SYSTEM Example System
  (* Version 1.0, 2007-08-28, Goran, Chalmers *)
  DEVICE Test Device : DeviceType_not_used
    RESOURCE TestResource : ResourceType_not_used
      FBS
        restart : E_RESTART;
        stop : E_STOP;
        split : E_SPLIT2;
        rend : E_REND;
        prod1 : Product;
        prod2 : Product;
        res1 : Resource;
        res2 : Resource;
        res3 : Resource;
        mux1take : Mux;
        mux1process : Mux;
        mux1release : Mux;
        mux2take : Mux;
        mux2process : Mux;
        mux2release : Mux;
        mux3take : Mux;
        mux3process : Mux;
        mux3release : Mux;
        datamux1 : DataMux;
        datamux2 : DataMux;
        datamux3 : DataMux;
        datademux1 : DataDemux;
        datademux2 : DataDemux;
        datademux3 : DataDemux;
        demux1taken : Demux;
        demux1processed : Demux;
        demux2taken : Demux;
        demux2processed : Demux;
        demux3taken : Demux;
        demux3processed : Demux;
      END_FBS
      EVENT_CONNECTIONS
        restart.COLD TO split.EI;
        split.EO1 TO prod1.make;
        split.EO2 TO prod2.make;
        prod1.takeR1 TO mux1take.EI1;
        prod1.processR1 TO mux1process.EI1;
        prod1.releaseR1 TO mux1release.EI1;
        prod2.takeR1 TO mux1take.EI2;
        prod2.processR1 TO mux1process.EI2;
        prod2.releaseR1 TO mux1release.EI2;
        mux1take.EO TO datamux1.EI1;
        mux1process.EO TO datamux1.EI2;
        mux1release.EO TO datamux1.EI3;
        datamux1.EO1 TO res1.take;
        datamux1.EO2 TO res1.process;
        datamux1.EO3 TO res1.release;
        res1.taken TO datademux1.EI1;
        res1.processed TO datademux1.EI2;
        datademux1.EO1 TO demux1taken.EI;
        datademux1.EO2 TO demux1processed.EI;
        demux1taken.EO1 TO prod1.gotR1;
        demux1taken.EO2 TO prod2.gotR1;
        demux1processed.EO1 TO prod1.processedR1;
        demux1processed.EO2 TO prod2.processedR1;
        prod1.takeR2 TO mux2take.EI1;
        prod1.processR2 TO mux2process.EI1;
        prod1.releaseR2 TO mux2release.EI1;
        prod2.takeR2 TO mux2take.EI2;
        prod2.processR2 TO mux2process.EI2;
        prod2.releaseR2 TO mux2release.EI2;
        mux2take.EO TO datamux2.EI1;
        mux2process.EO TO datamux2.EI2;
        mux2release.EO TO datamux2.EI3;
        datamux2.EO1 TO res2.take;
        datamux2.EO2 TO res2.process;
        datamux2.EO3 TO res2.release;
        res2.taken TO datademux2.EI1;
        res2.processed TO datademux2.EI2;
        datademux2.EO1 TO demux2taken.EI;
        datademux2.EO2 TO demux2processed.EI;
        demux2taken.EO1 TO prod1.gotR2;
        demux2taken.EO2 TO prod2.gotR2;
        demux2processed.EO1 TO prod1.processedR2;
        demux2processed.EO2 TO prod2.processedR2;
        prod1.takeR3 TO mux3take.EI1;
        prod1.processR3 TO mux3process.EI1;
        prod1.releaseR3 TO mux3release.EI1;
        prod2.takeR3 TO mux3take.EI2;
        prod2.processR3 TO mux3process.EI2;
        prod2.releaseR3 TO mux3release.EI2;
        mux3take.EO TO datamux3.EI1;
        mux3process.EO TO datamux3.EI2;
        mux3release.EO TO datamux3.EI3;
        datamux3.EO1 TO res3.take;
        datamux3.EO2 TO res3.process;
        datamux3.EO3 TO res3.release;
        res3.taken TO datademux3.EI1;
        res3.processed TO datademux3.EI2;
        datademux3.EO1 TO demux3taken.EI;
        datademux3.EO2 TO demux3processed.EI;
        demux3taken.EO1 TO prod1.gotR3;
        demux3taken.EO2 TO prod2.gotR3;
        demux3processed.EO1 TO prod1.processedR3;
        demux3processed.EO2 TO prod2.processedR3;
        prod1.done TO rend.EI1;
        prod2.done TO rend.EI2;
        rend.EO TO stop.STOP;
      END_CONNECTIONS
      DATA_CONNECTIONS
        1 TO prod1.product;
        2 TO prod2.product;
        1 TO res1.capacity;
        1 TO res2.capacity;
        1 TO res3.capacity;
        mux1take.DO TO datamux1.DI1;
        mux1process.DO TO datamux1.DI2;
        mux1release.DO TO datamux1.DI3;
        datamux1.DO TO res1.product;
        res1.forProduct TO datademux1.DI;
        datademux1.DO1 TO demux1taken.DI;
        datademux1.DO2 TO demux1processed.DI;
        mux2take.DO TO datamux2.DI1;
        mux2process.DO TO datamux2.DI2;
        mux2release.DO TO datamux2.DI3;
        datamux2.DO TO res2.product;
        res2.forProduct TO datademux2.DI;
        datademux2.DO1 TO demux2taken.DI;
        datademux2.DO2 TO demux2processed.DI;
        mux3take.DO TO datamux3.DI1;
        mux3process.DO TO datamux3.DI2;
        mux3release.DO TO datamux3.DI3;
        datamux3.DO TO res3.product;
        res3.forProduct TO datademux3.DI;
        datademux3.DO1 TO demux3taken.DI;
        datademux3.DO2 TO demux3processed.DI;
      END_CONNECTIONS
    END_RESOURCE
  END_DEVICE
END_SYSTEM
